FUNCTION_BLOCK POU EXTENDS FB_Contactor IMPLEMENTS I_DriveDouble
VAR_INPUT
END_VAR
VAR_OUTPUT
END_VAR
VAR
END_VAR

{error 'add property implementation or delete property to use base implementation'}
PROPERTY AutoToggle : BOOL
GET
END_GET
SET
END_SET
END_PROPERTY

{error 'add method implementation or delete method to use base implementation'}
METHOD SwitchForwardOff : BOOL
END_METHOD

{error 'add method implementation or delete method to use base implementation'}
METHOD SwitchForwardOn : BOOL
END_METHOD

{warning 'add method implementation '}
METHOD SwitchReverseOff : BOOL
END_METHOD

{warning 'add method implementation '}
METHOD SwitchReverseOn : BOOL
END_METHOD

END_FUNCTION_BLOCK

(* stored: Version 1.1.0.1, ProductVersion 3.1.4024.12
   POU POU: Id {48133537-34d4-4612-9e66-963ba226311c}, SpecialFunc None
   Property AutoToggle: Id {8bdcf332-6957-439d-927d-839c98f5dabc}
   Get Get: Id {08bee13e-0e88-4b31-b70f-c1fa56739221}
   Set Set: Id {bd0ca6ca-89cd-4e98-9b49-42e2a189e267}
   Method SwitchForwardOff: Id {f890c330-467d-4bec-9b9e-d627684caade}
   Method SwitchForwardOn: Id {9a97f4fd-9acd-4ef1-9321-6b4c876412f7}
   Method SwitchReverseOff: Id {76edae8d-ef50-4496-8d51-35c20281e523}
   Method SwitchReverseOn: Id {d432c05b-2341-4086-bd0d-b577d7d674c6} *)
